// TIA Portal V15.1 export
// export: Created 2024-05-17T05:38:44.5507069Z, ExportSetting WithDefaults, DisplayName Totally Integrated Automation Portal, DisplayVersion V15.1 Update 5, DisplayName TIA Portal Openness, DisplayVersion V15.1 Update 5, DisplayName SINAMICS Startdrive Advanced, DisplayVersion V15.1, DisplayName G130, G150, S120, S150, SINAMICS MV, S210, DisplayVersion V15.1, DisplayName G110M, G120, G120C, G120D, G120P, DisplayVersion V15.1, DisplayName STEP 7 Professional, DisplayVersion V15.1 Update 5, DisplayName STEP 7 Safety, DisplayVersion V15.1, DisplayName WinCC Professional, DisplayVersion V15.1 Update 5, DisplayName SIMATIC Visualization Architect, DisplayVersion V15.1
FUNCTION_BLOCK "LGBStackLight"   // FB6680, FBD
TITLE = LGBStackLight
{ S7_Optimized_Access := 'TRUE' }
VERSION : 0.1
// =============================================================================
// This module handles indication for Start, Alarm Reset.
// =============================================================================
// stored: AutoNumber false, IsIECCheckEnabled false, IsRetainMemResEnabled false, MemoryReserve 100, SetENOAutomatically False, UDAEnableTagReadback false
   VAR_INPUT
      I_ResetSafetyActive { ExternalAccessible := 'False'; ExternalVisible := 'False'; ExternalWritable := 'False'} : Bool;   // Reset of safety is active
   END_VAR
   VAR_OUTPUT
      O_AutoInd { ExternalAccessible := 'False'; ExternalVisible := 'False'; ExternalWritable := 'False'} : Bool;   // Auto lamp indication
      O_AlarmInd { ExternalAccessible := 'False'; ExternalVisible := 'False'; ExternalWritable := 'False'} : Bool;   // Alarm lamp Indication
      O_Buzzer { ExternalAccessible := 'False'; ExternalVisible := 'False'; ExternalWritable := 'False'} : Bool;
   END_VAR
   VAR_IN_OUT
      IO_ModesZM1 : "Modes";   // Modes ZM1
      IO_ModesZM2 : "Modes";   // Modes ZM2
      IO_ModesZM3 : "Modes";   // Modes ZM3
      IO_ModesZM4 : "Modes";   // Modes ZM4
      IO_ModesZM5 : "Modes";   // Modes ZM5
      IO_ModesZM6 : "Modes";   // Modes ZM6
      IO_ModesZM7 : "Modes";   // Modes ZM7
      IO_ModesZM8 : "Modes";   // Modes ZM8
      IO_ModesZM9 : "Modes";   // Modes ZM9
      IO_ModesZM10 : "Modes";   // Modes ZM10
      IO_ModesZM11 : "Modes";   // Modes ZM11
      IO_ModesZM12 : "Modes";   // Modes ZM12
      IO_ModesZM13 : "Modes";   // Modes ZM13
      IO_ModesZM14 : "Modes";   // Modes ZM14
      IO_ModesZM15 : "Modes";   // Modes ZM15
      IO_ModesZM16 : "Modes";   // Modes ZM16
   END_VAR
   VAR
      ZMAlarmLampSteadyCondition { ExternalAccessible := 'False'; ExternalVisible := 'False'; ExternalWritable := 'False'} : Bool;   // Alarm conditions active
      ZSAlarmLampSteadyCondition { ExternalAccessible := 'False'; ExternalVisible := 'False'; ExternalWritable := 'False'} : Bool;   // Alarm conditions active
      PLCAlarmLampSteadyCondition { ExternalAccessible := 'False'; ExternalVisible := 'False'; ExternalWritable := 'False'} : Bool;   // Alarm conditions active
      SafetyOk { ExternalAccessible := 'False'; ExternalVisible := 'False'; ExternalWritable := 'False'} : Bool;   // SafetyOk / No Haltbutton is activate
      Lamptest { ExternalAccessible := 'False'; ExternalVisible := 'False'; ExternalWritable := 'False'} : Bool;   // Lamptest selected alternating signal
      LamptestSteady { ExternalAccessible := 'False'; ExternalVisible := 'False'; ExternalWritable := 'False'} : Bool;   // Lamptest selected steady signal
      AutoModeSelected { ExternalAccessible := 'False'; ExternalVisible := 'False'; ExternalWritable := 'False'} : Bool;   // Automatic mode selected
      AutoMode { ExternalAccessible := 'False'; ExternalVisible := 'False'; ExternalWritable := 'False'} : Bool;   // Automatic mode active
      AutoInd { ExternalAccessible := 'False'; ExternalVisible := 'False'; ExternalWritable := 'False'} : Bool;   // Auto indication
      AlarmInd { ExternalAccessible := 'False'; ExternalVisible := 'False'; ExternalWritable := 'False'} : Bool;   // Alarm Indication
      BuzzzerCond { ExternalAccessible := 'False'; ExternalVisible := 'False'; ExternalWritable := 'False'} : Bool;   // Buzzer activation conditins
   END_VAR
BEGIN

REGION Network 1: **** 4.2 - Machine status - Calculated **** ZM level Alarm condition AB active
   // Alarm condition AB active
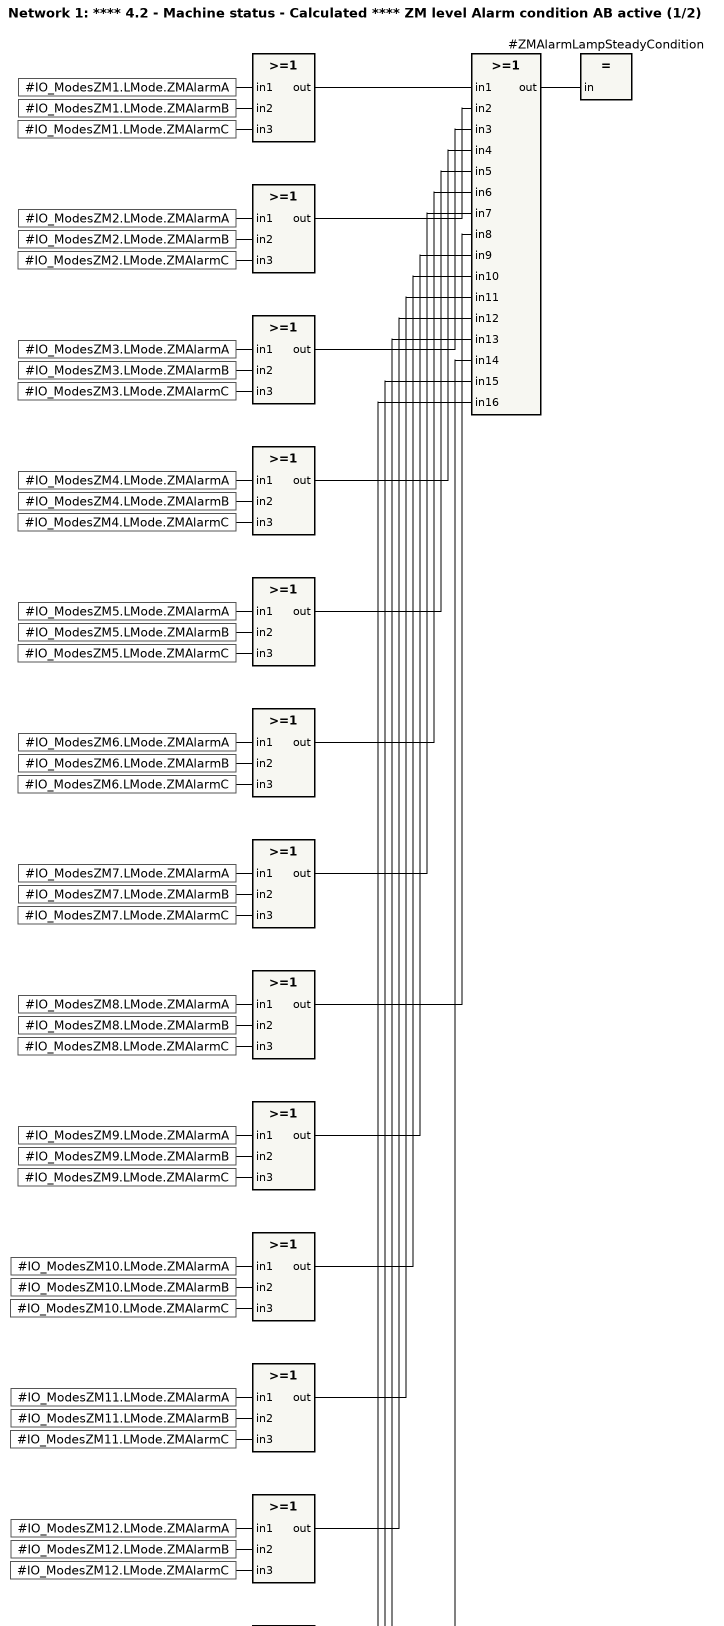
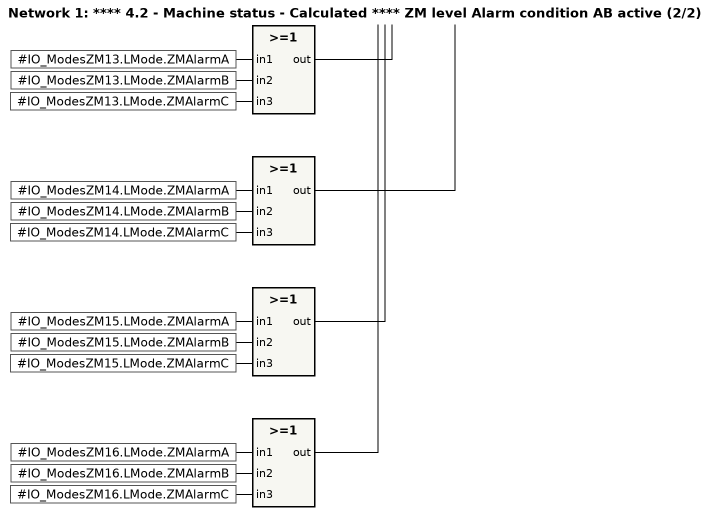
   #ZMAlarmLampSteadyCondition := #IO_ModesZM1.LMode.ZMAlarmA OR #IO_ModesZM1.LMode.ZMAlarmB OR #IO_ModesZM1.LMode.ZMAlarmC OR #IO_ModesZM2.LMode.ZMAlarmA OR #IO_ModesZM2.LMode.ZMAlarmB OR #IO_ModesZM2.LMode.ZMAlarmC OR #IO_ModesZM3.LMode.ZMAlarmA OR #IO_ModesZM3.LMode.ZMAlarmB OR #IO_ModesZM3.LMode.ZMAlarmC OR #IO_ModesZM4.LMode.ZMAlarmA OR #IO_ModesZM4.LMode.ZMAlarmB OR #IO_ModesZM4.LMode.ZMAlarmC OR #IO_ModesZM5.LMode.ZMAlarmA OR #IO_ModesZM5.LMode.ZMAlarmB OR #IO_ModesZM5.LMode.ZMAlarmC OR #IO_ModesZM6.LMode.ZMAlarmA OR #IO_ModesZM6.LMode.ZMAlarmB OR #IO_ModesZM6.LMode.ZMAlarmC OR #IO_ModesZM7.LMode.ZMAlarmA OR #IO_ModesZM7.LMode.ZMAlarmB OR #IO_ModesZM7.LMode.ZMAlarmC OR #IO_ModesZM8.LMode.ZMAlarmA OR #IO_ModesZM8.LMode.ZMAlarmB OR #IO_ModesZM8.LMode.ZMAlarmC OR #IO_ModesZM9.LMode.ZMAlarmA OR #IO_ModesZM9.LMode.ZMAlarmB OR #IO_ModesZM9.LMode.ZMAlarmC OR #IO_ModesZM10.LMode.ZMAlarmA OR #IO_ModesZM10.LMode.ZMAlarmB OR #IO_ModesZM10.LMode.ZMAlarmC OR #IO_ModesZM11.LMode.ZMAlarmA OR #IO_ModesZM11.LMode.ZMAlarmB OR #IO_ModesZM11.LMode.ZMAlarmC OR #IO_ModesZM12.LMode.ZMAlarmA OR #IO_ModesZM12.LMode.ZMAlarmB OR #IO_ModesZM12.LMode.ZMAlarmC OR #IO_ModesZM13.LMode.ZMAlarmA OR #IO_ModesZM13.LMode.ZMAlarmB OR #IO_ModesZM13.LMode.ZMAlarmC OR #IO_ModesZM14.LMode.ZMAlarmA OR #IO_ModesZM14.LMode.ZMAlarmB OR #IO_ModesZM14.LMode.ZMAlarmC OR #IO_ModesZM15.LMode.ZMAlarmA OR #IO_ModesZM15.LMode.ZMAlarmB OR #IO_ModesZM15.LMode.ZMAlarmC OR #IO_ModesZM16.LMode.ZMAlarmA OR #IO_ModesZM16.LMode.ZMAlarmB OR #IO_ModesZM16.LMode.ZMAlarmC;
END_REGION

REGION Network 2: **** 4.2 - Machine status - Calculated **** ZS level Alarm condition AB active
   // Alarm condition AB active
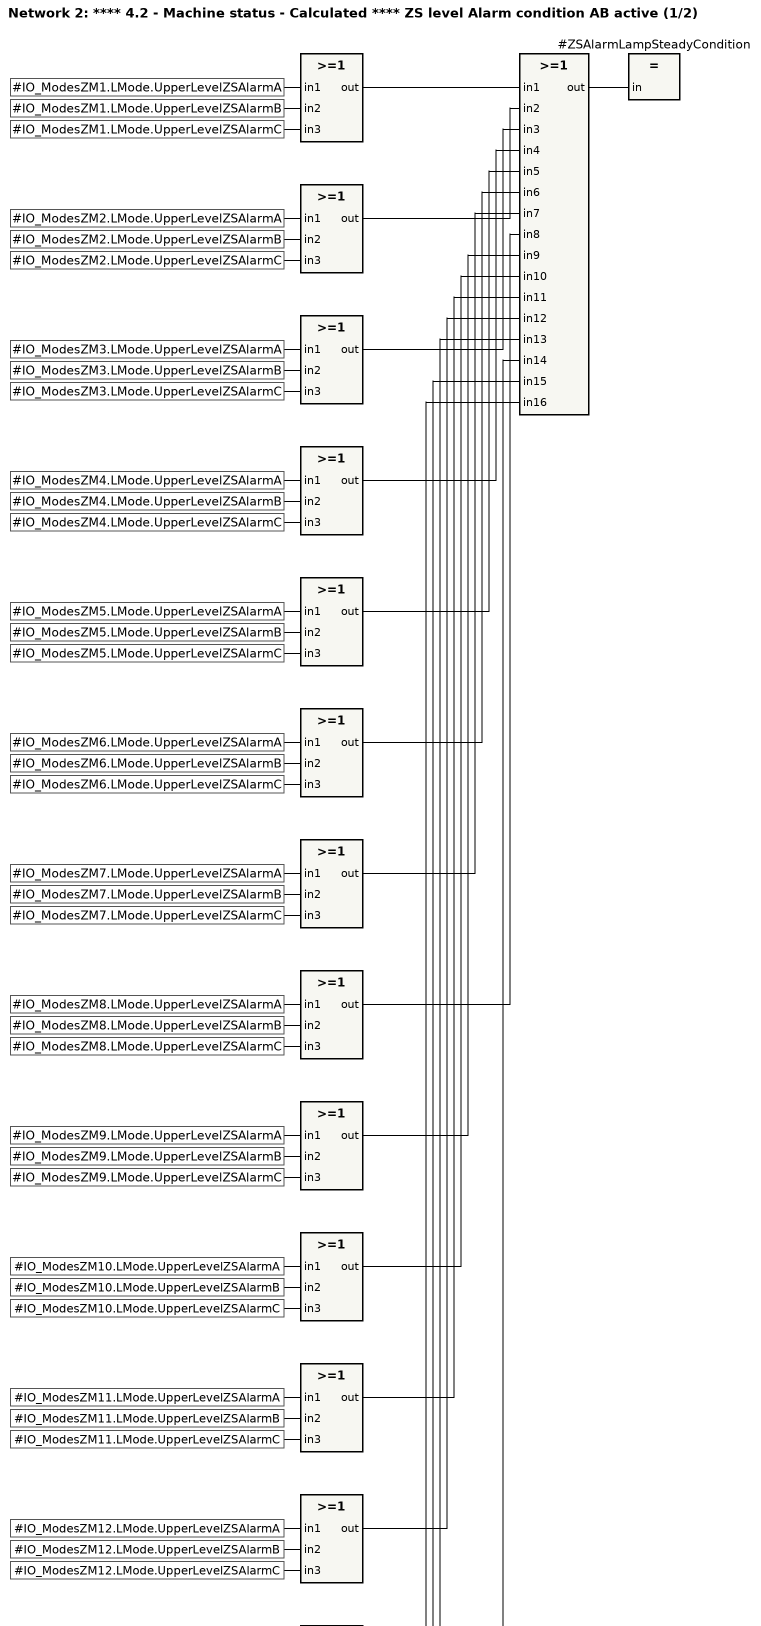
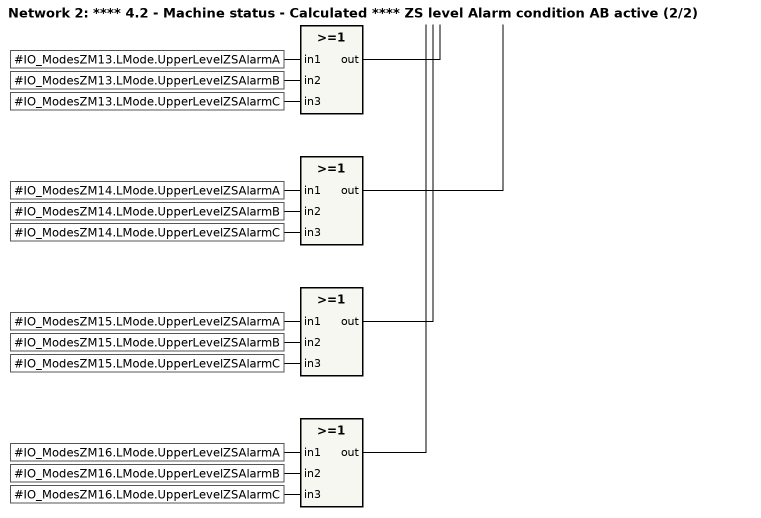
   #ZSAlarmLampSteadyCondition := #IO_ModesZM1.LMode.UpperLevelZSAlarmA OR #IO_ModesZM1.LMode.UpperLevelZSAlarmB OR #IO_ModesZM1.LMode.UpperLevelZSAlarmC OR #IO_ModesZM2.LMode.UpperLevelZSAlarmA OR #IO_ModesZM2.LMode.UpperLevelZSAlarmB OR #IO_ModesZM2.LMode.UpperLevelZSAlarmC OR #IO_ModesZM3.LMode.UpperLevelZSAlarmA OR #IO_ModesZM3.LMode.UpperLevelZSAlarmB OR #IO_ModesZM3.LMode.UpperLevelZSAlarmC OR #IO_ModesZM4.LMode.UpperLevelZSAlarmA OR #IO_ModesZM4.LMode.UpperLevelZSAlarmB OR #IO_ModesZM4.LMode.UpperLevelZSAlarmC OR #IO_ModesZM5.LMode.UpperLevelZSAlarmA OR #IO_ModesZM5.LMode.UpperLevelZSAlarmB OR #IO_ModesZM5.LMode.UpperLevelZSAlarmC OR #IO_ModesZM6.LMode.UpperLevelZSAlarmA OR #IO_ModesZM6.LMode.UpperLevelZSAlarmB OR #IO_ModesZM6.LMode.UpperLevelZSAlarmC OR #IO_ModesZM7.LMode.UpperLevelZSAlarmA OR #IO_ModesZM7.LMode.UpperLevelZSAlarmB OR #IO_ModesZM7.LMode.UpperLevelZSAlarmC OR #IO_ModesZM8.LMode.UpperLevelZSAlarmA OR #IO_ModesZM8.LMode.UpperLevelZSAlarmB OR #IO_ModesZM8.LMode.UpperLevelZSAlarmC OR #IO_ModesZM9.LMode.UpperLevelZSAlarmA OR #IO_ModesZM9.LMode.UpperLevelZSAlarmB OR #IO_ModesZM9.LMode.UpperLevelZSAlarmC OR #IO_ModesZM10.LMode.UpperLevelZSAlarmA OR #IO_ModesZM10.LMode.UpperLevelZSAlarmB OR #IO_ModesZM10.LMode.UpperLevelZSAlarmC OR #IO_ModesZM11.LMode.UpperLevelZSAlarmA OR #IO_ModesZM11.LMode.UpperLevelZSAlarmB OR #IO_ModesZM11.LMode.UpperLevelZSAlarmC OR #IO_ModesZM12.LMode.UpperLevelZSAlarmA OR #IO_ModesZM12.LMode.UpperLevelZSAlarmB OR #IO_ModesZM12.LMode.UpperLevelZSAlarmC OR #IO_ModesZM13.LMode.UpperLevelZSAlarmA OR #IO_ModesZM13.LMode.UpperLevelZSAlarmB OR #IO_ModesZM13.LMode.UpperLevelZSAlarmC OR #IO_ModesZM14.LMode.UpperLevelZSAlarmA OR #IO_ModesZM14.LMode.UpperLevelZSAlarmB OR #IO_ModesZM14.LMode.UpperLevelZSAlarmC OR #IO_ModesZM15.LMode.UpperLevelZSAlarmA OR #IO_ModesZM15.LMode.UpperLevelZSAlarmB OR #IO_ModesZM15.LMode.UpperLevelZSAlarmC OR #IO_ModesZM16.LMode.UpperLevelZSAlarmA OR #IO_ModesZM16.LMode.UpperLevelZSAlarmB OR #IO_ModesZM16.LMode.UpperLevelZSAlarmC;
END_REGION

REGION Network 3: **** 4.2 - Machine status - Calculated **** PLC level Alarm condition AB active
   // Alarm condition AB active
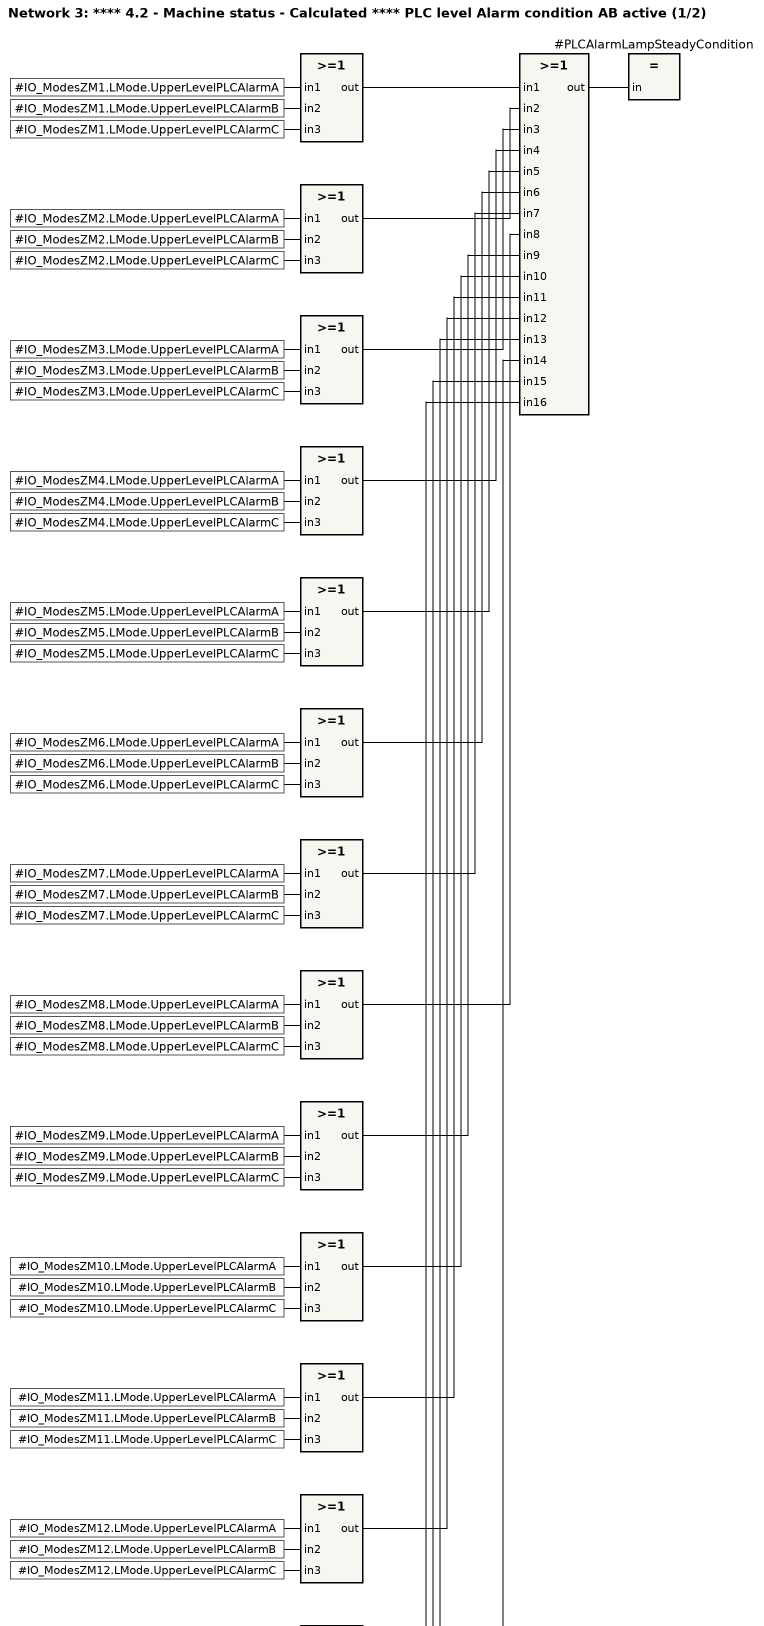
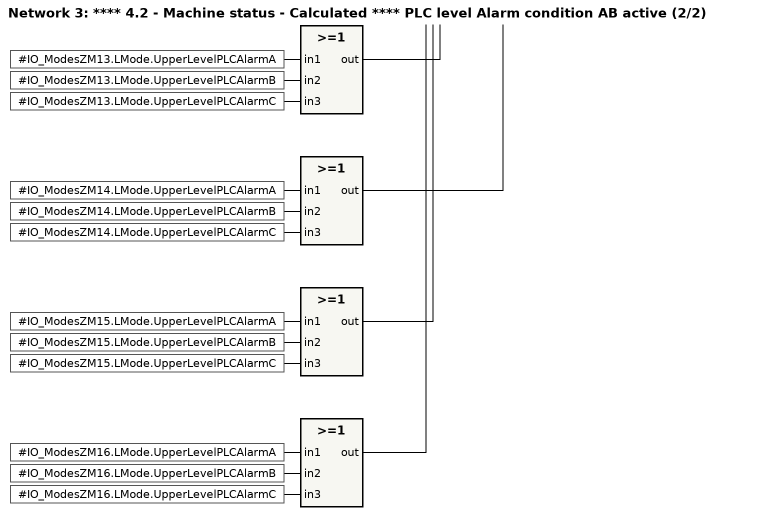
   #PLCAlarmLampSteadyCondition := #IO_ModesZM1.LMode.UpperLevelPLCAlarmA OR #IO_ModesZM1.LMode.UpperLevelPLCAlarmB OR #IO_ModesZM1.LMode.UpperLevelPLCAlarmC OR #IO_ModesZM2.LMode.UpperLevelPLCAlarmA OR #IO_ModesZM2.LMode.UpperLevelPLCAlarmB OR #IO_ModesZM2.LMode.UpperLevelPLCAlarmC OR #IO_ModesZM3.LMode.UpperLevelPLCAlarmA OR #IO_ModesZM3.LMode.UpperLevelPLCAlarmB OR #IO_ModesZM3.LMode.UpperLevelPLCAlarmC OR #IO_ModesZM4.LMode.UpperLevelPLCAlarmA OR #IO_ModesZM4.LMode.UpperLevelPLCAlarmB OR #IO_ModesZM4.LMode.UpperLevelPLCAlarmC OR #IO_ModesZM5.LMode.UpperLevelPLCAlarmA OR #IO_ModesZM5.LMode.UpperLevelPLCAlarmB OR #IO_ModesZM5.LMode.UpperLevelPLCAlarmC OR #IO_ModesZM6.LMode.UpperLevelPLCAlarmA OR #IO_ModesZM6.LMode.UpperLevelPLCAlarmB OR #IO_ModesZM6.LMode.UpperLevelPLCAlarmC OR #IO_ModesZM7.LMode.UpperLevelPLCAlarmA OR #IO_ModesZM7.LMode.UpperLevelPLCAlarmB OR #IO_ModesZM7.LMode.UpperLevelPLCAlarmC OR #IO_ModesZM8.LMode.UpperLevelPLCAlarmA OR #IO_ModesZM8.LMode.UpperLevelPLCAlarmB OR #IO_ModesZM8.LMode.UpperLevelPLCAlarmC OR #IO_ModesZM9.LMode.UpperLevelPLCAlarmA OR #IO_ModesZM9.LMode.UpperLevelPLCAlarmB OR #IO_ModesZM9.LMode.UpperLevelPLCAlarmC OR #IO_ModesZM10.LMode.UpperLevelPLCAlarmA OR #IO_ModesZM10.LMode.UpperLevelPLCAlarmB OR #IO_ModesZM10.LMode.UpperLevelPLCAlarmC OR #IO_ModesZM11.LMode.UpperLevelPLCAlarmA OR #IO_ModesZM11.LMode.UpperLevelPLCAlarmB OR #IO_ModesZM11.LMode.UpperLevelPLCAlarmC OR #IO_ModesZM12.LMode.UpperLevelPLCAlarmA OR #IO_ModesZM12.LMode.UpperLevelPLCAlarmB OR #IO_ModesZM12.LMode.UpperLevelPLCAlarmC OR #IO_ModesZM13.LMode.UpperLevelPLCAlarmA OR #IO_ModesZM13.LMode.UpperLevelPLCAlarmB OR #IO_ModesZM13.LMode.UpperLevelPLCAlarmC OR #IO_ModesZM14.LMode.UpperLevelPLCAlarmA OR #IO_ModesZM14.LMode.UpperLevelPLCAlarmB OR #IO_ModesZM14.LMode.UpperLevelPLCAlarmC OR #IO_ModesZM15.LMode.UpperLevelPLCAlarmA OR #IO_ModesZM15.LMode.UpperLevelPLCAlarmB OR #IO_ModesZM15.LMode.UpperLevelPLCAlarmC OR #IO_ModesZM16.LMode.UpperLevelPLCAlarmA OR #IO_ModesZM16.LMode.UpperLevelPLCAlarmB OR #IO_ModesZM16.LMode.UpperLevelPLCAlarmC;
END_REGION

REGION Network 4: **** 4.2 - Machine status - Calculated **** Safety Ok
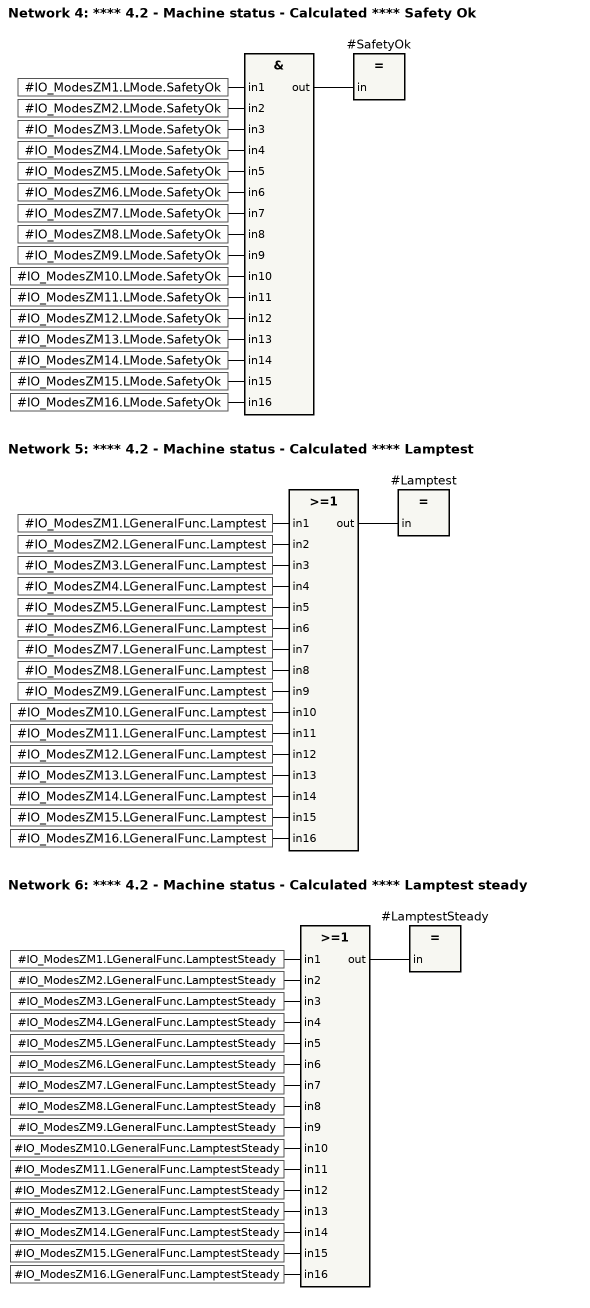
   #SafetyOk := #IO_ModesZM1.LMode.SafetyOk AND #IO_ModesZM2.LMode.SafetyOk AND #IO_ModesZM3.LMode.SafetyOk AND #IO_ModesZM4.LMode.SafetyOk AND #IO_ModesZM5.LMode.SafetyOk AND #IO_ModesZM6.LMode.SafetyOk AND #IO_ModesZM7.LMode.SafetyOk AND #IO_ModesZM8.LMode.SafetyOk AND #IO_ModesZM9.LMode.SafetyOk AND #IO_ModesZM10.LMode.SafetyOk AND #IO_ModesZM11.LMode.SafetyOk AND #IO_ModesZM12.LMode.SafetyOk AND #IO_ModesZM13.LMode.SafetyOk AND #IO_ModesZM14.LMode.SafetyOk AND #IO_ModesZM15.LMode.SafetyOk AND #IO_ModesZM16.LMode.SafetyOk;
END_REGION

REGION Network 5: **** 4.2 - Machine status - Calculated **** Lamptest
   // Lamptest
   #Lamptest := #IO_ModesZM1.LGeneralFunc.Lamptest OR #IO_ModesZM2.LGeneralFunc.Lamptest OR #IO_ModesZM3.LGeneralFunc.Lamptest OR #IO_ModesZM4.LGeneralFunc.Lamptest OR #IO_ModesZM5.LGeneralFunc.Lamptest OR #IO_ModesZM6.LGeneralFunc.Lamptest OR #IO_ModesZM7.LGeneralFunc.Lamptest OR #IO_ModesZM8.LGeneralFunc.Lamptest OR #IO_ModesZM9.LGeneralFunc.Lamptest OR #IO_ModesZM10.LGeneralFunc.Lamptest OR #IO_ModesZM11.LGeneralFunc.Lamptest OR #IO_ModesZM12.LGeneralFunc.Lamptest OR #IO_ModesZM13.LGeneralFunc.Lamptest OR #IO_ModesZM14.LGeneralFunc.Lamptest OR #IO_ModesZM15.LGeneralFunc.Lamptest OR #IO_ModesZM16.LGeneralFunc.Lamptest;
END_REGION

REGION Network 6: **** 4.2 - Machine status - Calculated **** Lamptest steady
   // Lamptest
   #LamptestSteady := #IO_ModesZM1.LGeneralFunc.LamptestSteady OR #IO_ModesZM2.LGeneralFunc.LamptestSteady OR #IO_ModesZM3.LGeneralFunc.LamptestSteady OR #IO_ModesZM4.LGeneralFunc.LamptestSteady OR #IO_ModesZM5.LGeneralFunc.LamptestSteady OR #IO_ModesZM6.LGeneralFunc.LamptestSteady OR #IO_ModesZM7.LGeneralFunc.LamptestSteady OR #IO_ModesZM8.LGeneralFunc.LamptestSteady OR #IO_ModesZM9.LGeneralFunc.LamptestSteady OR #IO_ModesZM10.LGeneralFunc.LamptestSteady OR #IO_ModesZM11.LGeneralFunc.LamptestSteady OR #IO_ModesZM12.LGeneralFunc.LamptestSteady OR #IO_ModesZM13.LGeneralFunc.LamptestSteady OR #IO_ModesZM14.LGeneralFunc.LamptestSteady OR #IO_ModesZM15.LGeneralFunc.LamptestSteady OR #IO_ModesZM16.LGeneralFunc.LamptestSteady;
END_REGION

REGION Network 7: **** 4.2 - Machine status - Calculated **** Automatic mode selected
   // Automatic mode selected
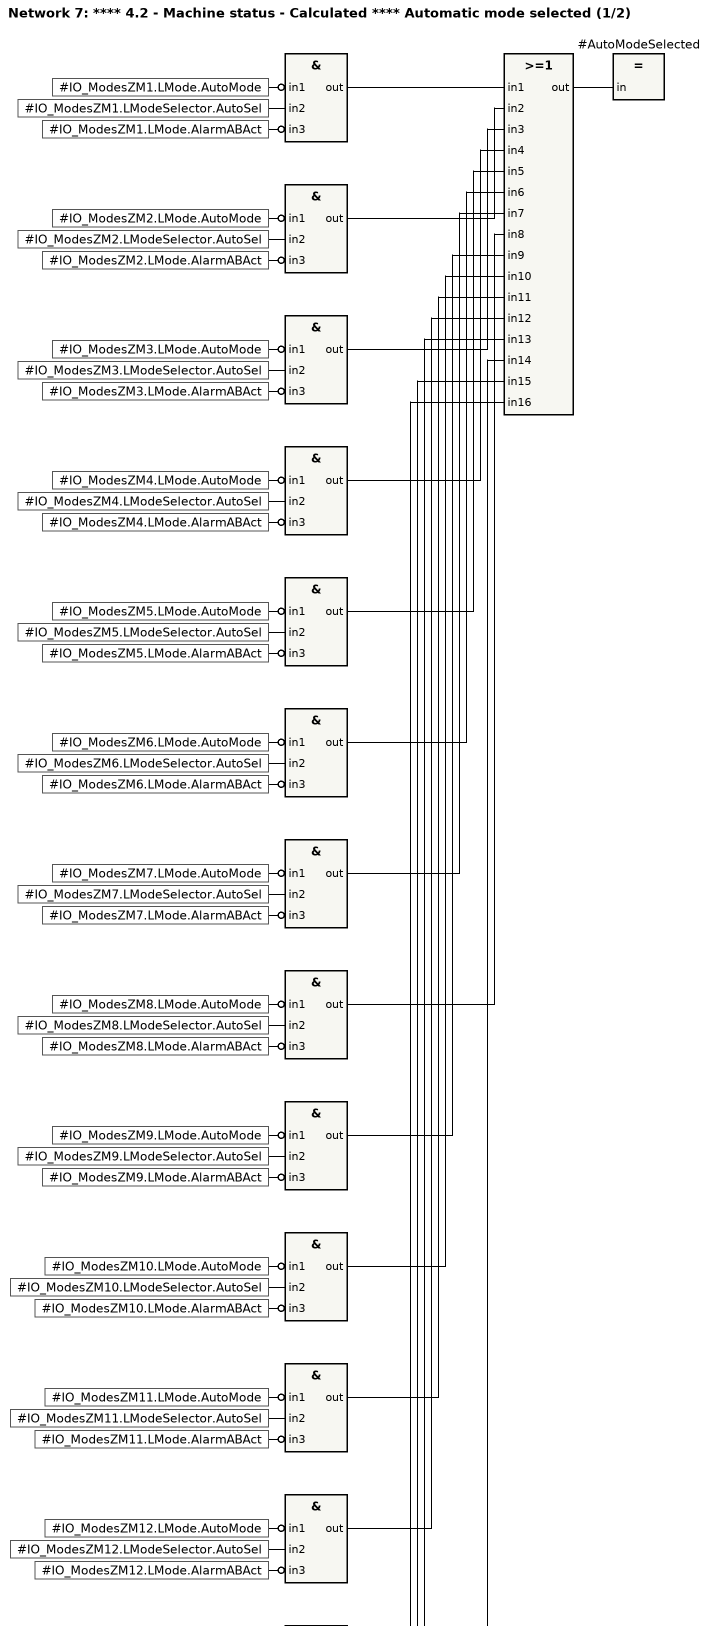
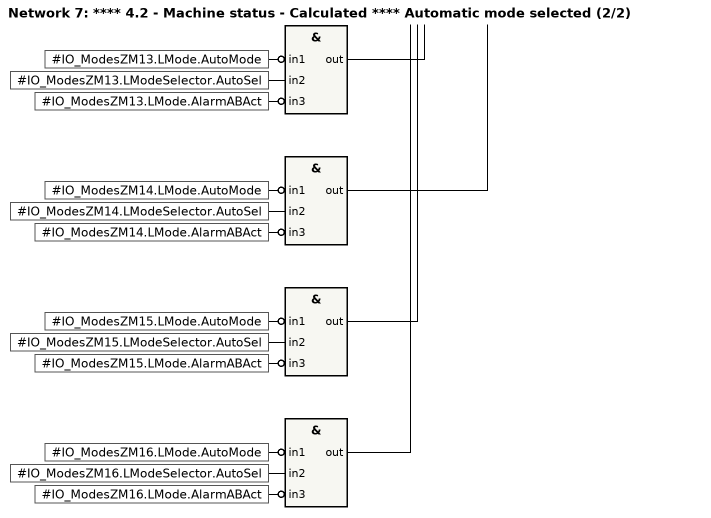
   #AutoModeSelected := (NOT #IO_ModesZM1.LMode.AutoMode AND #IO_ModesZM1.LModeSelector.AutoSel AND NOT #IO_ModesZM1.LMode.AlarmABAct) OR (NOT #IO_ModesZM2.LMode.AutoMode AND #IO_ModesZM2.LModeSelector.AutoSel AND NOT #IO_ModesZM2.LMode.AlarmABAct) OR (NOT #IO_ModesZM3.LMode.AutoMode AND #IO_ModesZM3.LModeSelector.AutoSel AND NOT #IO_ModesZM3.LMode.AlarmABAct) OR (NOT #IO_ModesZM4.LMode.AutoMode AND #IO_ModesZM4.LModeSelector.AutoSel AND NOT #IO_ModesZM4.LMode.AlarmABAct) OR (NOT #IO_ModesZM5.LMode.AutoMode AND #IO_ModesZM5.LModeSelector.AutoSel AND NOT #IO_ModesZM5.LMode.AlarmABAct) OR (NOT #IO_ModesZM6.LMode.AutoMode AND #IO_ModesZM6.LModeSelector.AutoSel AND NOT #IO_ModesZM6.LMode.AlarmABAct) OR (NOT #IO_ModesZM7.LMode.AutoMode AND #IO_ModesZM7.LModeSelector.AutoSel AND NOT #IO_ModesZM7.LMode.AlarmABAct) OR (NOT #IO_ModesZM8.LMode.AutoMode AND #IO_ModesZM8.LModeSelector.AutoSel AND NOT #IO_ModesZM8.LMode.AlarmABAct) OR (NOT #IO_ModesZM9.LMode.AutoMode AND #IO_ModesZM9.LModeSelector.AutoSel AND NOT #IO_ModesZM9.LMode.AlarmABAct) OR (NOT #IO_ModesZM10.LMode.AutoMode AND #IO_ModesZM10.LModeSelector.AutoSel AND NOT #IO_ModesZM10.LMode.AlarmABAct) OR (NOT #IO_ModesZM11.LMode.AutoMode AND #IO_ModesZM11.LModeSelector.AutoSel AND NOT #IO_ModesZM11.LMode.AlarmABAct) OR (NOT #IO_ModesZM12.LMode.AutoMode AND #IO_ModesZM12.LModeSelector.AutoSel AND NOT #IO_ModesZM12.LMode.AlarmABAct) OR (NOT #IO_ModesZM13.LMode.AutoMode AND #IO_ModesZM13.LModeSelector.AutoSel AND NOT #IO_ModesZM13.LMode.AlarmABAct) OR (NOT #IO_ModesZM14.LMode.AutoMode AND #IO_ModesZM14.LModeSelector.AutoSel AND NOT #IO_ModesZM14.LMode.AlarmABAct) OR (NOT #IO_ModesZM15.LMode.AutoMode AND #IO_ModesZM15.LModeSelector.AutoSel AND NOT #IO_ModesZM15.LMode.AlarmABAct) OR (NOT #IO_ModesZM16.LMode.AutoMode AND #IO_ModesZM16.LModeSelector.AutoSel AND NOT #IO_ModesZM16.LMode.AlarmABAct);
END_REGION

REGION Network 8: **** 4.2 - Machine status - Calculated **** Automatic mode active
   // Automatic mode active
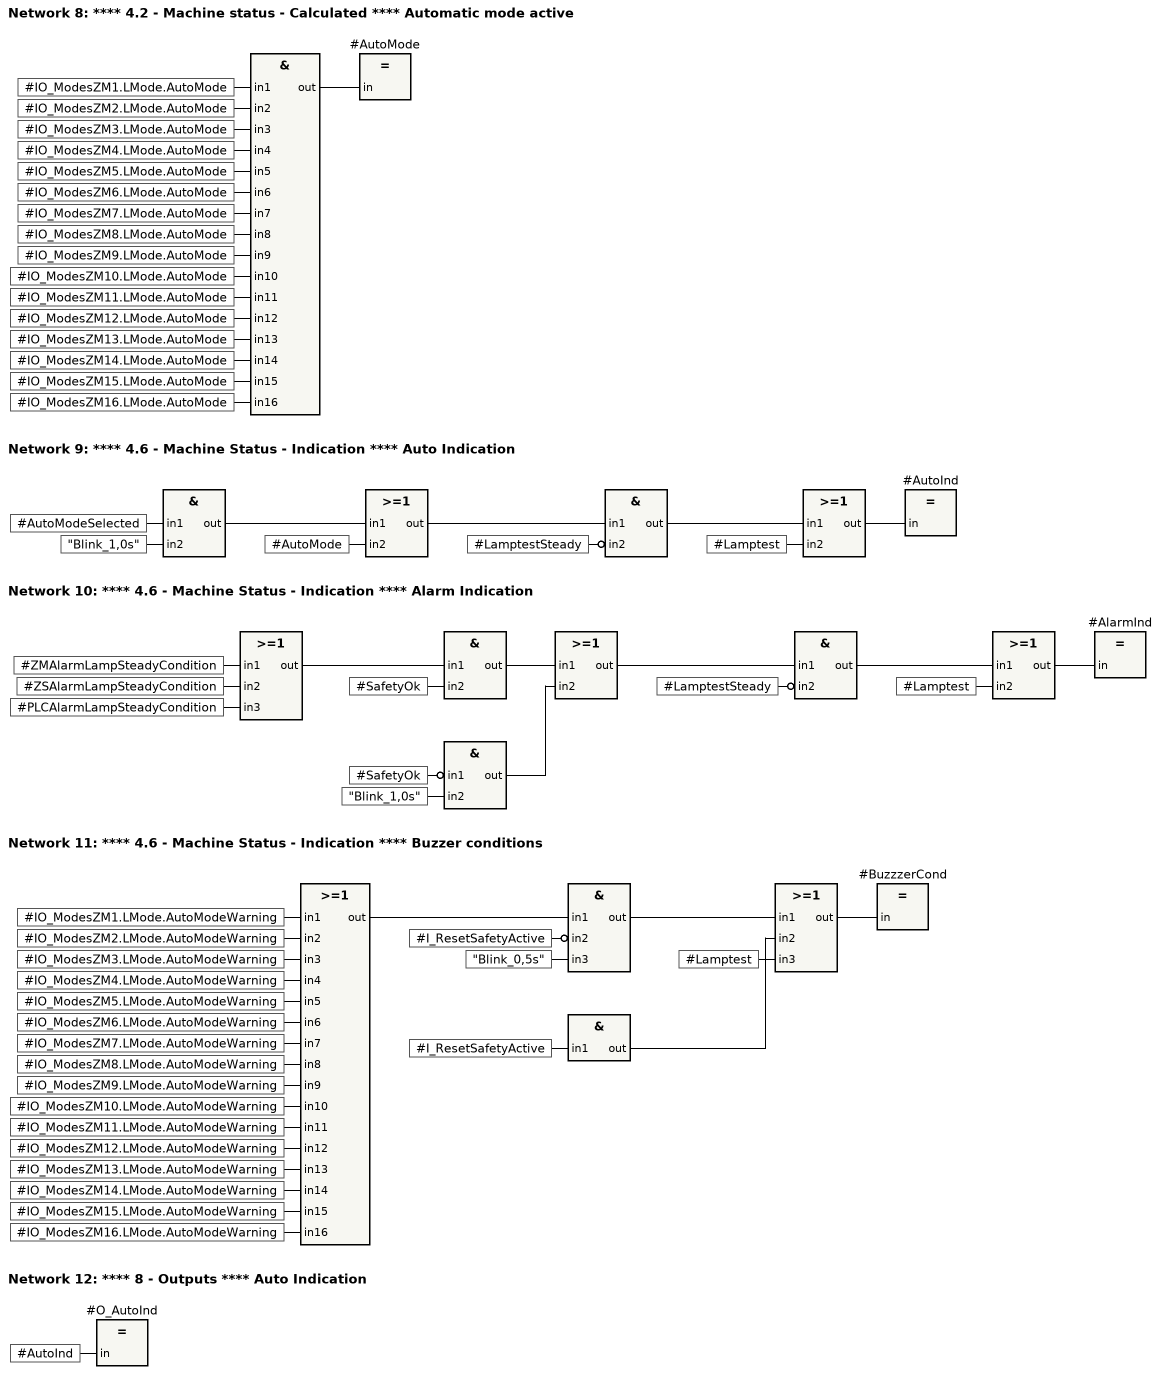
   #AutoMode := #IO_ModesZM1.LMode.AutoMode AND #IO_ModesZM2.LMode.AutoMode AND #IO_ModesZM3.LMode.AutoMode AND #IO_ModesZM4.LMode.AutoMode AND #IO_ModesZM5.LMode.AutoMode AND #IO_ModesZM6.LMode.AutoMode AND #IO_ModesZM7.LMode.AutoMode AND #IO_ModesZM8.LMode.AutoMode AND #IO_ModesZM9.LMode.AutoMode AND #IO_ModesZM10.LMode.AutoMode AND #IO_ModesZM11.LMode.AutoMode AND #IO_ModesZM12.LMode.AutoMode AND #IO_ModesZM13.LMode.AutoMode AND #IO_ModesZM14.LMode.AutoMode AND #IO_ModesZM15.LMode.AutoMode AND #IO_ModesZM16.LMode.AutoMode;
END_REGION

REGION Network 9: **** 4.6 - Machine Status - Indication **** Auto Indication
   // Auto indication
   #AutoInd := (((#AutoModeSelected AND "Blink_1,0s") OR #AutoMode) AND NOT #LamptestSteady) OR #Lamptest;
END_REGION

REGION Network 10: **** 4.6 - Machine Status - Indication **** Alarm Indication
   // Alarm indication
   #AlarmInd := ((((#ZMAlarmLampSteadyCondition OR #ZSAlarmLampSteadyCondition OR #PLCAlarmLampSteadyCondition) AND #SafetyOk) OR (NOT #SafetyOk AND "Blink_1,0s")) AND NOT #LamptestSteady) OR #Lamptest;
END_REGION

REGION Network 11: **** 4.6 - Machine Status - Indication **** Buzzer conditions
   #BuzzzerCond := ((#IO_ModesZM1.LMode.AutoModeWarning OR #IO_ModesZM2.LMode.AutoModeWarning OR #IO_ModesZM3.LMode.AutoModeWarning OR #IO_ModesZM4.LMode.AutoModeWarning OR #IO_ModesZM5.LMode.AutoModeWarning OR #IO_ModesZM6.LMode.AutoModeWarning OR #IO_ModesZM7.LMode.AutoModeWarning OR #IO_ModesZM8.LMode.AutoModeWarning OR #IO_ModesZM9.LMode.AutoModeWarning OR #IO_ModesZM10.LMode.AutoModeWarning OR #IO_ModesZM11.LMode.AutoModeWarning OR #IO_ModesZM12.LMode.AutoModeWarning OR #IO_ModesZM13.LMode.AutoModeWarning OR #IO_ModesZM14.LMode.AutoModeWarning OR #IO_ModesZM15.LMode.AutoModeWarning OR #IO_ModesZM16.LMode.AutoModeWarning) AND NOT #I_ResetSafetyActive AND "Blink_0,5s") OR #I_ResetSafetyActive OR #Lamptest;
END_REGION

REGION Network 12: **** 8 - Outputs **** Auto Indication
   // Alarm Indication
   #O_AutoInd := #AutoInd;
END_REGION

REGION Network 13: **** 8 - Outputs **** Alarm Indication
   // Alarm Indication
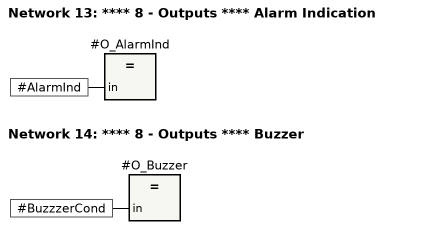
   #O_AlarmInd := #AlarmInd;
END_REGION

REGION Network 14: **** 8 - Outputs **** Buzzer
   // Buzzer conditions
   #O_Buzzer := #BuzzzerCond;
END_REGION
END_FUNCTION_BLOCK
